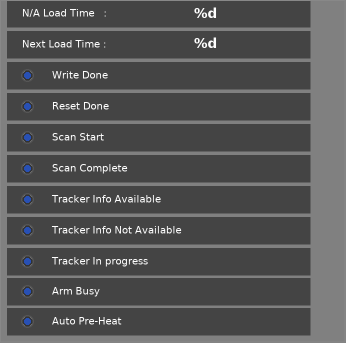
VISUALIZATION Popup_OtherInfo  // 346x343
    Rectangle (0,0 346x343)
    Rectangle (7,0 303x27)
    Label (19,1 100x24), "N/A Load Time :"
    Rectangle (7,31 303x27)
    Label (19,32 104x24), "Next Load Time :"
    Rectangle (7,62 303x27)
    Label (49,63 259x24), "Write Done"
    Lamp1 (20,68 15x15), variable: bMTBWriteDoneFlag, style: Lamp-Lamp1-Blue
    Rectangle (7,93 303x27)
    Label (49,94 258x24), "Reset Done"
    Lamp1 (20,99 15x15), variable: bMTBResetDoneFlag, style: Lamp-Lamp1-Blue
    Rectangle (7,124 303x27)
    Label (49,125 257x24), "Scan Start"
    Lamp1 (20,130 15x15), variable: bMTBScanEn AND NOT.bCallRTB_NoTrackerInfo, style: Lamp-Lamp1-Blue
    Rectangle (7,155 303x27)
    Label (49,156 256x24), "Scan Complete"
    Lamp1 (20,161 15x15), variable: bMTBScanCompletedFlag, style: Lamp-Lamp1-Blue
    Rectangle (7,186 303x27)
    Label (49,187 256x24), "Tracker Info Available"
    Lamp1 (20,192 15x15), variable: bCallRTB_CallOK, style: Lamp-Lamp1-Blue
    Rectangle (7,217 303x27)
    Label (49,218 259x24), "Tracker Info Not Available"
    Lamp1 (20,223 15x15), variable: bCallRTB_NoTrackerInfo, style: Lamp-Lamp1-Blue
    Rectangle (7,248 303x27)
    Label (49,249 257x24), "Tracker In progress"
    Lamp1 (20,254 15x15), variable: bTrackerStartEN, style: Lamp-Lamp1-Blue
    Rectangle (7,278 303x27)
    Label (49,279 256x24), "Arm Busy"
    Lamp1 (20,284 15x15), variable: ARbMTBArmProgress[1], style: Lamp-Lamp1-Blue
    Rectangle (7,308 303x27)
    Label (49,309 256x24), "Auto Pre-Heat"
    Lamp1 (20,314 15x15), variable: .bAutoPreparationPb AND NOT.bAutoPreparationDone, style: Lamp-Lamp1-Blue
    Rectangle (121,5 169x17), "%d", text variable: iMTBNextNotAvailableTime
    Rectangle (121,35 169x17), "%d", text variable: iMTBNextTransferTime
END_VISUALIZATION

(* stored: Version 1.1.0.1, ProductVersion 3.1.4024.12
   Visu Popup_OtherInfo: Id {a18718f0-7079-4419-a4aa-a8226262aa8c} *)
